// Mitsubishi GX Works2 project: אוטומציה 29.11 713   PLC: FX3G

// global labels: Global1
VAR_GLOBAL
  startDay AT X010 : BOOL;
  flourContainer AT D1110 : REAL;
  flourInput AT D1100 : REAL;
  yeastInput AT D1102 : REAL;
  yeatContainer AT D1112 : REAL;
  YeastContainer AT D1112 : REAL;
  waterInput AT D1104 : REAL;
  waterContainer AT D1114 : REAL;
  oilInput AT D1106 : REAL;
  oilContainer AT D1116 : REAL;
  spaicesInput AT D1108 : REAL;
  spaicesContainer AT D1118 : REAL;
  EmergencyStop AT X007 : BOOL;
  workDayLight AT Y010 : BOOL;
  endDay AT M8 : BOOL;
  outOfStock AT M7 : BOOL;
  startProduction AT M6 : BOOL;
END_VAR
VAR_GLOBAL CONSTANT
  minFlour : REAL := 100.0;
END_VAR
VAR_GLOBAL
  FlourOK AT M1 : BOOL;
END_VAR
VAR_GLOBAL CONSTANT
  fYratio : REAL := 0.2;
END_VAR
VAR_GLOBAL
  yeastOK AT M2 : BOOL;
END_VAR
VAR_GLOBAL CONSTANT
  wFratio : REAL := 0.5;
END_VAR
VAR_GLOBAL
  waterOK AT M3 : BOOL;
END_VAR
VAR_GLOBAL CONSTANT
  oFratio : REAL := 0.3;
END_VAR
VAR_GLOBAL
  oilOK AT M4 : BOOL;
END_VAR
VAR_GLOBAL CONSTANT
  sFratio : REAL := 0.1;
END_VAR
VAR_GLOBAL
  spaicesOK AT M5 : BOOL;
  LoadMaterialsButton AT X002 : BOOL;
  LoadMterialsLamp AT Y005 : BOOL;
END_VAR
VAR_GLOBAL CONSTANT
  flour_100 : REAL := 100;
  Yeast_20 : REAL := 20;
  water_50 : REAL := 50;
  oil_30 : REAL := 30;
  spices_10 : REAL := 10;
END_VAR
VAR_GLOBAL
  timeVal_3sec AT K30 : INT;
  prepTimer AT TC10 : BOOL;
  prepTimer_out AT TS10 : BOOL;
  startLisha AT X001 : BOOL;
  proofStartHatpaha AT M32 : BOOL;
  lishaMotor AT Y001 : BOOL;
  hatpaha_Counter AT CC1 : BOOL;
  doubleclick AT K2 : WORD;
  start_Hatpaha AT X011 : BOOL;
  outC1 AT CS1 : BOOL;
  y2timer AT TC22 : BOOL;
  TS22_out AT TS22 : BOOL;
  ind_blinkled AT M0 : BOOL;
  Hatpaha_led2 AT Y002 : BOOL;
  y3timer AT TC23 : BOOL;
  TS23_out AT TS23 : BOOL;
  Hatpaha_led3 AT Y003 : BOOL;
  hatpaha_timer AT TC32 : BOOL;
  TS32_OUT AT TS32 : BOOL;
  timeVal_BLINK AT K5 : INT;
  y4timer AT TC24 : BOOL;
  timeVal_4 AT K40 : INT;
  BAKE_LAMP AT Y004 : BOOL;
  TS24_out AT TS24 : BOOL;
  quality_check AT X003 : BOOL;
  Analog_Input_2 AT D8281 : INT;
  Save_analog_val AT D8201 : INT;
END_VAR
VAR_GLOBAL CONSTANT
  min_val : INT := 400;
  max_val : INT := 2000;
END_VAR
VAR_GLOBAL
  Analog_GT AT M11 : BOOL;
  Analog_LT AT M12 : BOOL;
  y6_timer AT TC26 : BOOL;
  timeVal_5 AT K50 : INT;
  TS26_out AT TS26 : BOOL;
  move_to_shelf_lamp AT Y006 : BOOL;
  check_counter AT CC2 : BOOL;
  double_check AT K2 : WORD;
  CC2_out AT CS2 : BOOL;
  batch_Rejact AT M23 : BOOL;
  in_Proportion AT M6 : BOOL;
END_VAR
VAR_GLOBAL CONSTANT
  iteration_Flour : INT := 100;
END_VAR
VAR_GLOBAL
  iteration_Flour_Container AT D1120 : REAL;
END_VAR
VAR_GLOBAL CONSTANT
  iteration_Flour_Amount : REAL := 100;
  iteration_Yeast_Amount : REAL := 20;
END_VAR
VAR_GLOBAL
  iteration_Yeast_Container AT D1122 : REAL;
END_VAR
VAR_GLOBAL CONSTANT
  iteration_Water_Amount : REAL := 50;
END_VAR
VAR_GLOBAL
  iteration_Water_Container AT D1124 : REAL;
END_VAR
VAR_GLOBAL CONSTANT
  iteration_Oil_Amount : REAL := 30;
END_VAR
VAR_GLOBAL
  iteration_Oil_Container AT D1126 : REAL;
END_VAR
VAR_GLOBAL CONSTANT
  iteration_Spices_Amount : REAL := 10;
END_VAR
VAR_GLOBAL
  iteration_Spices_Container AT D1128 : REAL;
  mearbel_container AT D1130 : REAL;
  hatpaha_Container AT D1132 : REAL;
  tavnit_bake_container AT D1134 : REAL;
  bakery_shelf_container AT D1136 : REAL;
  noFlour AT M40 : BOOL;
  noYeast AT M42 : BOOL;
  noWater AT M44 : BOOL;
  noOil AT M46 : BOOL;
  noSpices AT M48 : BOOL;
END_VAR
VAR_GLOBAL CONSTANT
  reset_0 : REAL;
END_VAR
VAR_GLOBAL
  finish_timer AT TC50 : BOOL;
  TS50_OUT AT TS50 : BOOL;
  ind_blinkled_finish AT M200 : BOOL;
  TS52_out AT TS52 : BOOL;
  TS54_out AT TS54 : BOOL;
  timeVal_BLINK2 AT K2 : INT;
  no_light_10 AT M60 : BOOL;
  end_day_light AT M62 : BOOL;
  ind AT M0 : BOOL;
  delete_mearbel AT M33 : BOOL;
  ind_move_to_tavnit AT M100 : BOOL;
  ind_move_to_bakery AT M102 : BOOL;
  y10blinkOn AT TC52 : BOOL;
  y10blinkOff AT TC54 : BOOL;
  y10_steady_light AT M70 : BOOL;
END_VAR
VAR_GLOBAL CONSTANT
  iteration_finished : REAL := 1;
END_VAR
VAR_GLOBAL
  ind_iteration_finished AT M250 : BOOL;
  ind_end_of_iteration AT M104 : BOOL;
  iteration_counter AT D1138 : REAL;
END_VAR
VAR_GLOBAL CONSTANT
  check_prev_lvl : REAL;
END_VAR
VAR_GLOBAL
  ind_first_lvl_finished AT M400 : BOOL;
  ind_X2_lvl_finished AT M402 : BOOL;
  ind_X11_lvl_finished AT M404 : BOOL;
END_VAR

// task Task_01 (event TRUE, interval 0, priority 31): POU_01

PROGRAM POU_01
(* structured ladder/FBD written out as ST: instructions are called as NAME(EN, inputs, outputs); _pN, _eN, _tN stand for wires *)
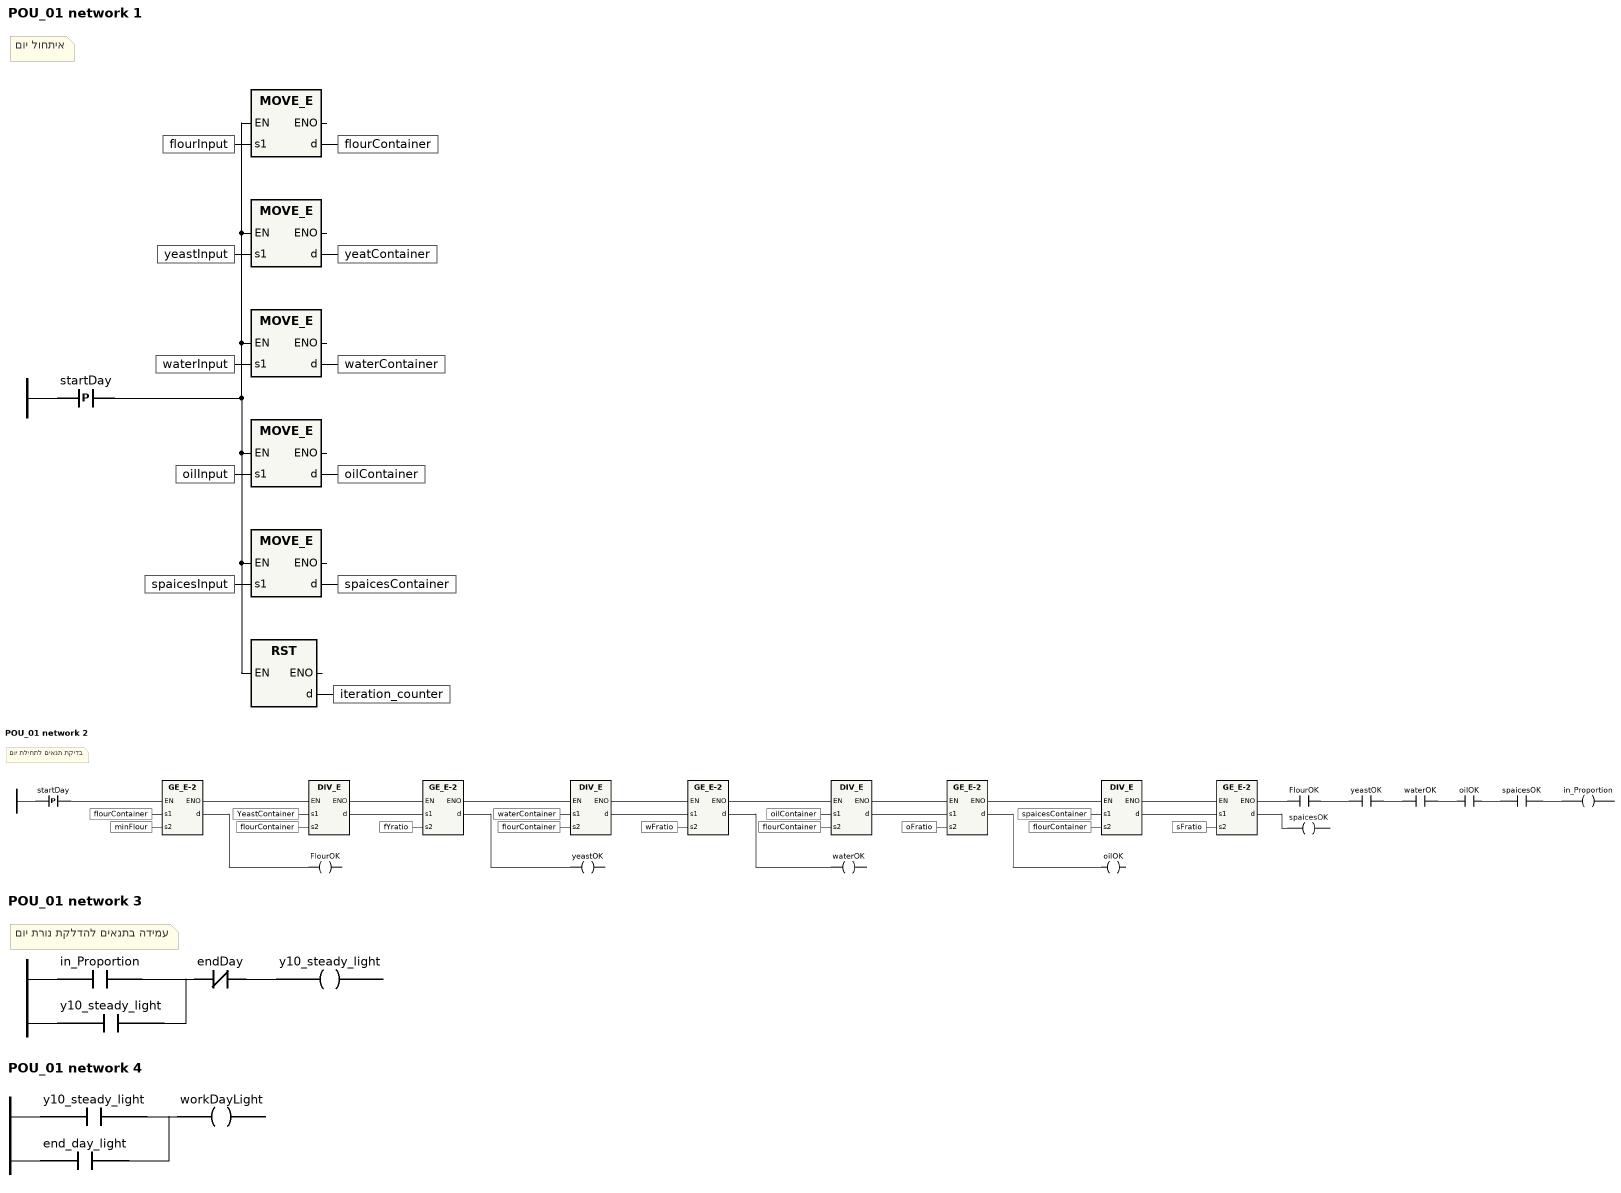
(* network 1 *)
(* איתחול יום *)
_p1 := LDP(TRUE, startDay);
MOVE_E(_p1, flourInput, flourContainer);
MOVE_E(_p1, yeastInput, yeatContainer);
MOVE_E(_p1, waterInput, waterContainer);
MOVE_E(_p1, oilInput, oilContainer);
MOVE_E(_p1, spaicesInput, spaicesContainer);
RST(_p1, iteration_counter);
(* network 2 *)
(* בדיקת תנאים לתחילת יום *)
_e2 := GE_E(LDP(TRUE, startDay), flourContainer, minFlour, _t1);
_e4 := DIV_E(_e2, YeastContainer, flourContainer, _t3);
_e6 := GE_E(_e4, _t3, fYratio, _t5);
_e8 := DIV_E(_e6, waterContainer, flourContainer, _t7);
_e10 := GE_E(_e8, _t7, wFratio, _t9);
_e12 := DIV_E(_e10, oilContainer, flourContainer, _t11);
_e14 := GE_E(_e12, _t11, oFratio, _t13);
_e16 := DIV_E(_e14, spaicesContainer, flourContainer, _t15);
_e18 := GE_E(_e16, _t15, sFratio, _t17);
in_Proportion := _e18 AND FlourOK AND yeastOK AND waterOK AND oilOK AND spaicesOK;
yeastOK := _t5;
waterOK := _t9;
oilOK := _t13;
spaicesOK := _t17;
FlourOK := _t1;
(* network 3 *)
(* עמידה בתנאים להדלקת נורת יום *)
y10_steady_light := (in_Proportion OR y10_steady_light) AND NOT endDay;
(* network 4 *)
workDayLight := y10_steady_light OR end_day_light;
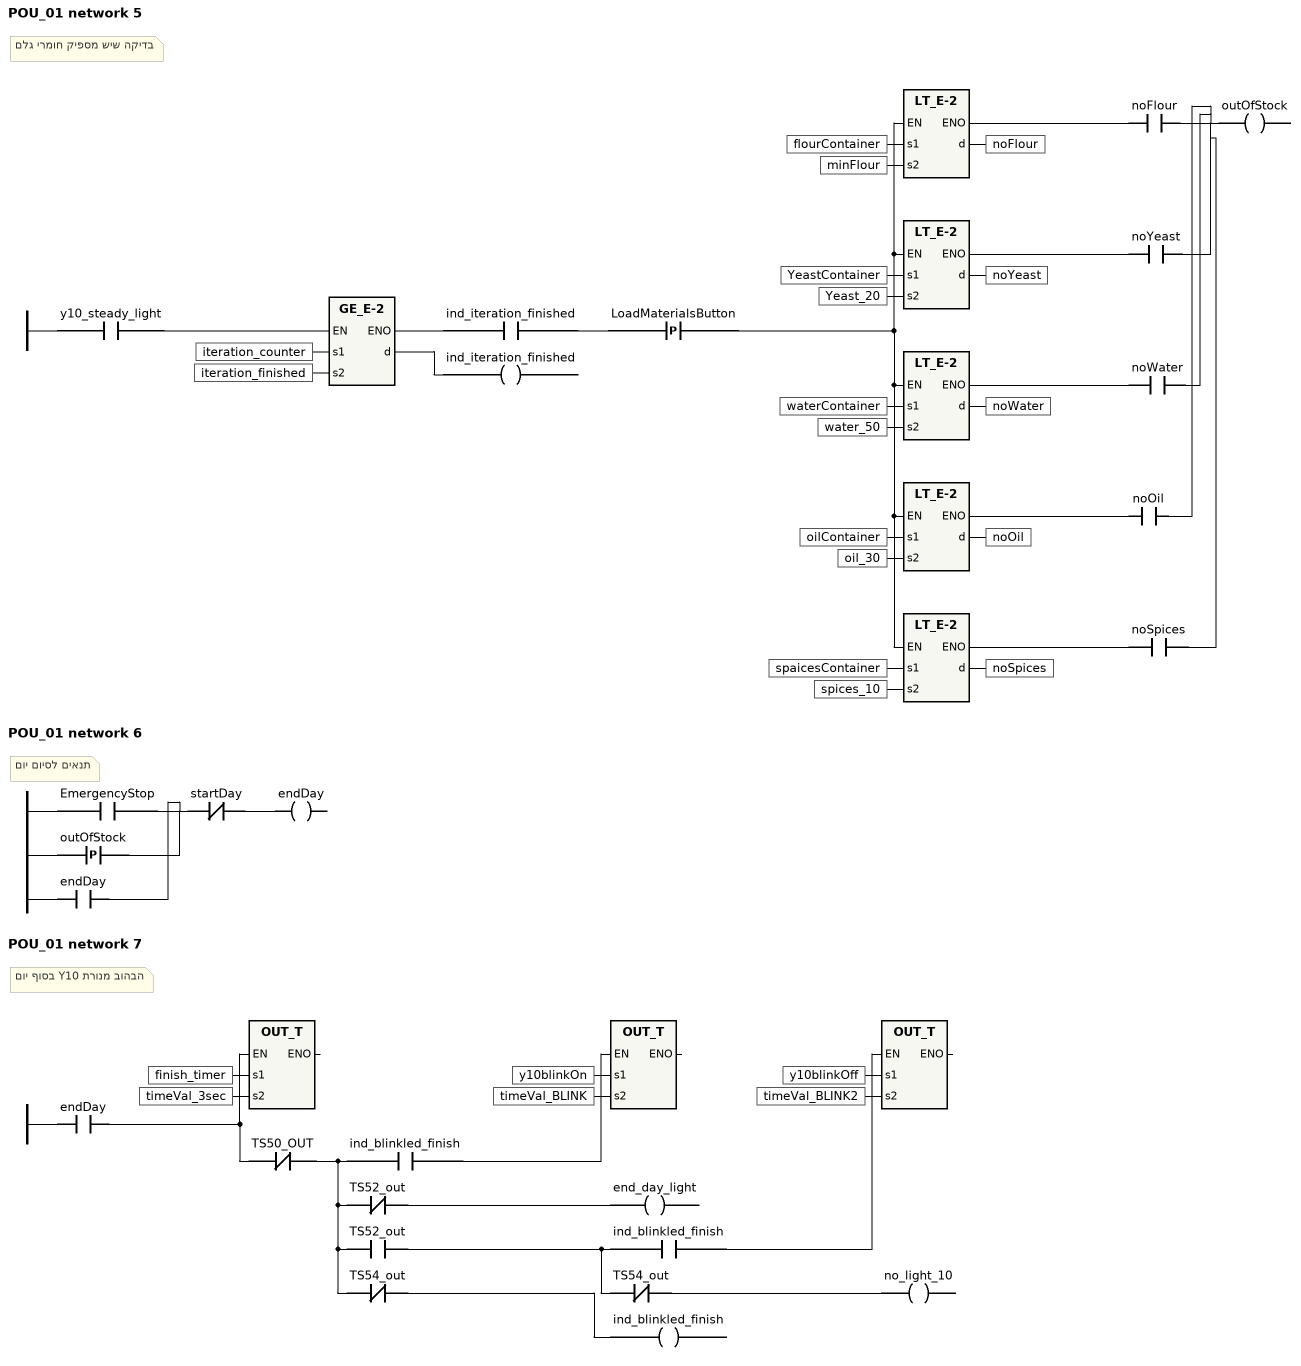
(* network 5 *)
(* בדיקה שיש מספיק חומרי גלם *)
_e2 := GE_E(y10_steady_light, iteration_counter, iteration_finished, _t1);
_p3 := _e2 AND ind_iteration_finished AND LDP(TRUE, LoadMaterialsButton);
_e4 := LT_E(_p3, flourContainer, minFlour, noFlour);
ind_iteration_finished := _t1;
_e5 := LT_E(_p3, YeastContainer, Yeast_20, noYeast);
_e6 := LT_E(_p3, waterContainer, water_50, noWater);
_e7 := LT_E(_p3, oilContainer, oil_30, noOil);
_e8 := LT_E(_p3, spaicesContainer, spices_10, noSpices);
outOfStock := (_e4 AND noFlour) OR (_e5 AND noYeast) OR (_e6 AND noWater) OR (_e7 AND noOil) OR (_e8 AND noSpices);
(* network 6 *)
(* תנאים לסיום יום *)
endDay := (EmergencyStop OR LDP(TRUE, outOfStock) OR endDay) AND NOT startDay;
(* network 7 *)
(* הבהוב מנורת Y10 בסוף יום *)
OUT_T(endDay, finish_timer, timeVal_3sec);
_p1 := endDay AND NOT TS50_OUT;
OUT_T(_p1 AND ind_blinkled_finish, y10blinkOn, timeVal_BLINK);
end_day_light := _p1 AND NOT TS52_out;
_p2 := _p1 AND TS52_out;
OUT_T(_p2 AND ind_blinkled_finish, y10blinkOff, timeVal_BLINK2);
no_light_10 := _p2 AND NOT TS54_out;
ind_blinkled_finish := _p1 AND NOT TS54_out;
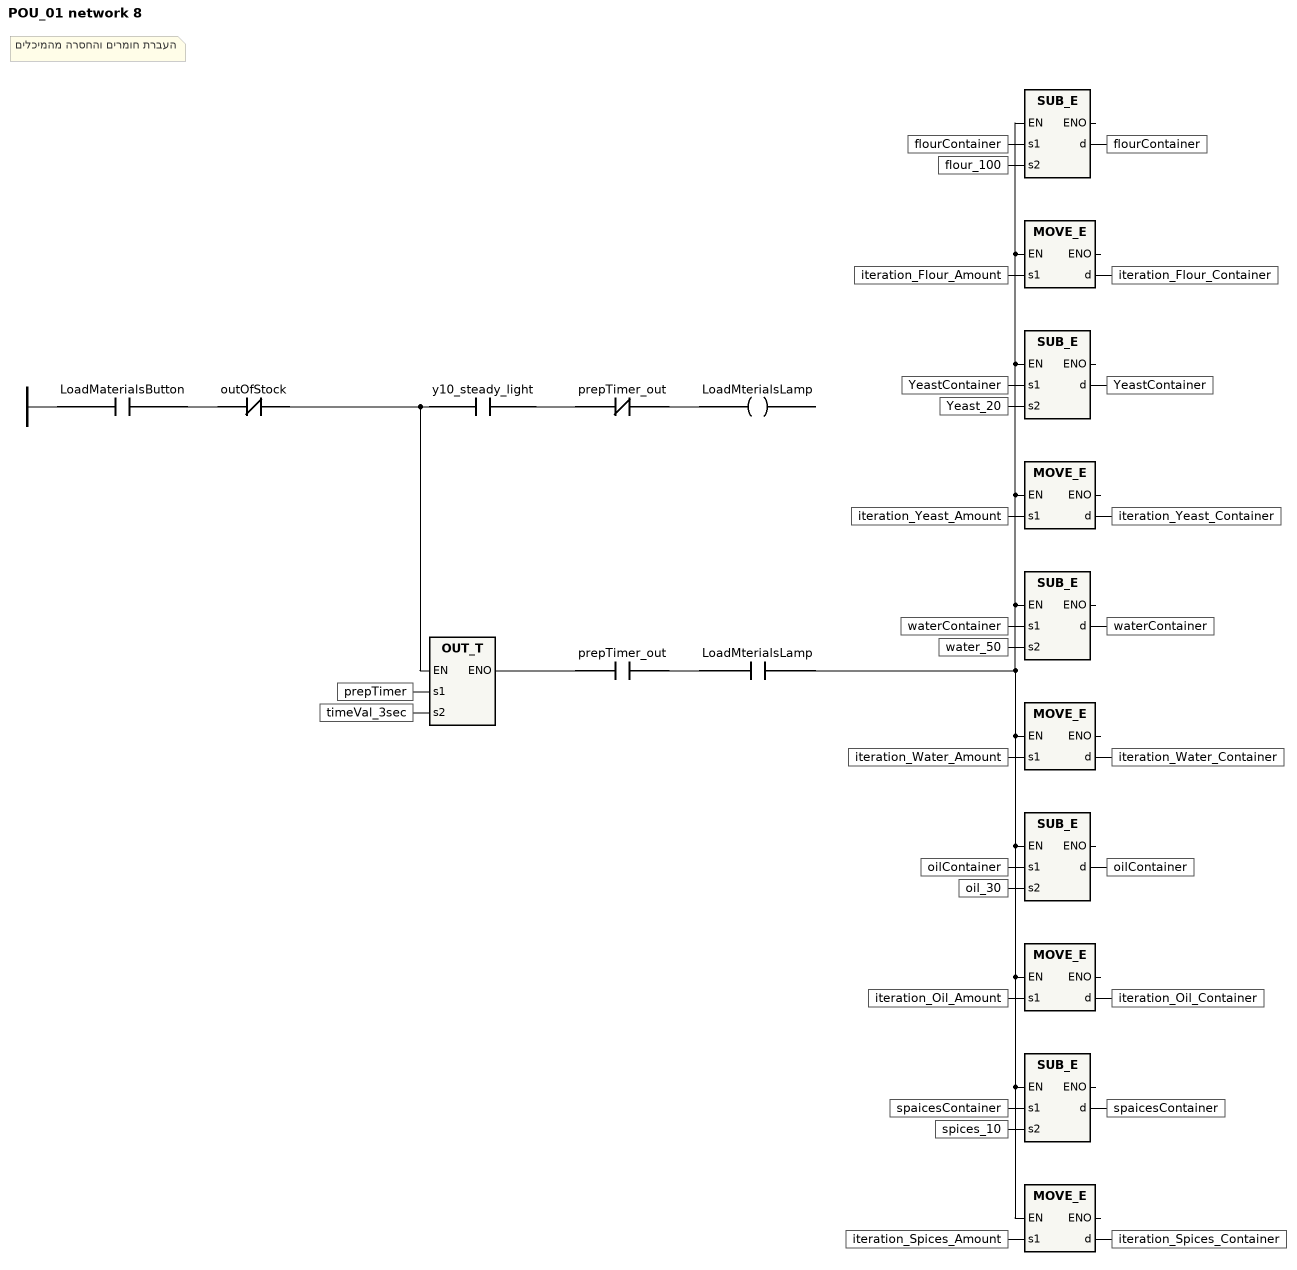
(* network 8 *)
(* העברת חומרים והחסרה מהמיכלים *)
_p1 := LoadMaterialsButton AND NOT outOfStock;
_e2 := OUT_T(_p1, prepTimer, timeVal_3sec);
_p3 := _e2 AND prepTimer_out AND LoadMterialsLamp;
SUB_E(_p3, flourContainer, flour_100, flourContainer);
MOVE_E(_p3, iteration_Flour_Amount, iteration_Flour_Container);
SUB_E(_p3, YeastContainer, Yeast_20, YeastContainer);
LoadMterialsLamp := _p1 AND y10_steady_light AND NOT prepTimer_out;
MOVE_E(_p3, iteration_Yeast_Amount, iteration_Yeast_Container);
SUB_E(_p3, waterContainer, water_50, waterContainer);
MOVE_E(_p3, iteration_Water_Amount, iteration_Water_Container);
SUB_E(_p3, oilContainer, oil_30, oilContainer);
MOVE_E(_p3, iteration_Oil_Amount, iteration_Oil_Container);
SUB_E(_p3, spaicesContainer, spices_10, spaicesContainer);
MOVE_E(_p3, iteration_Spices_Amount, iteration_Spices_Container);
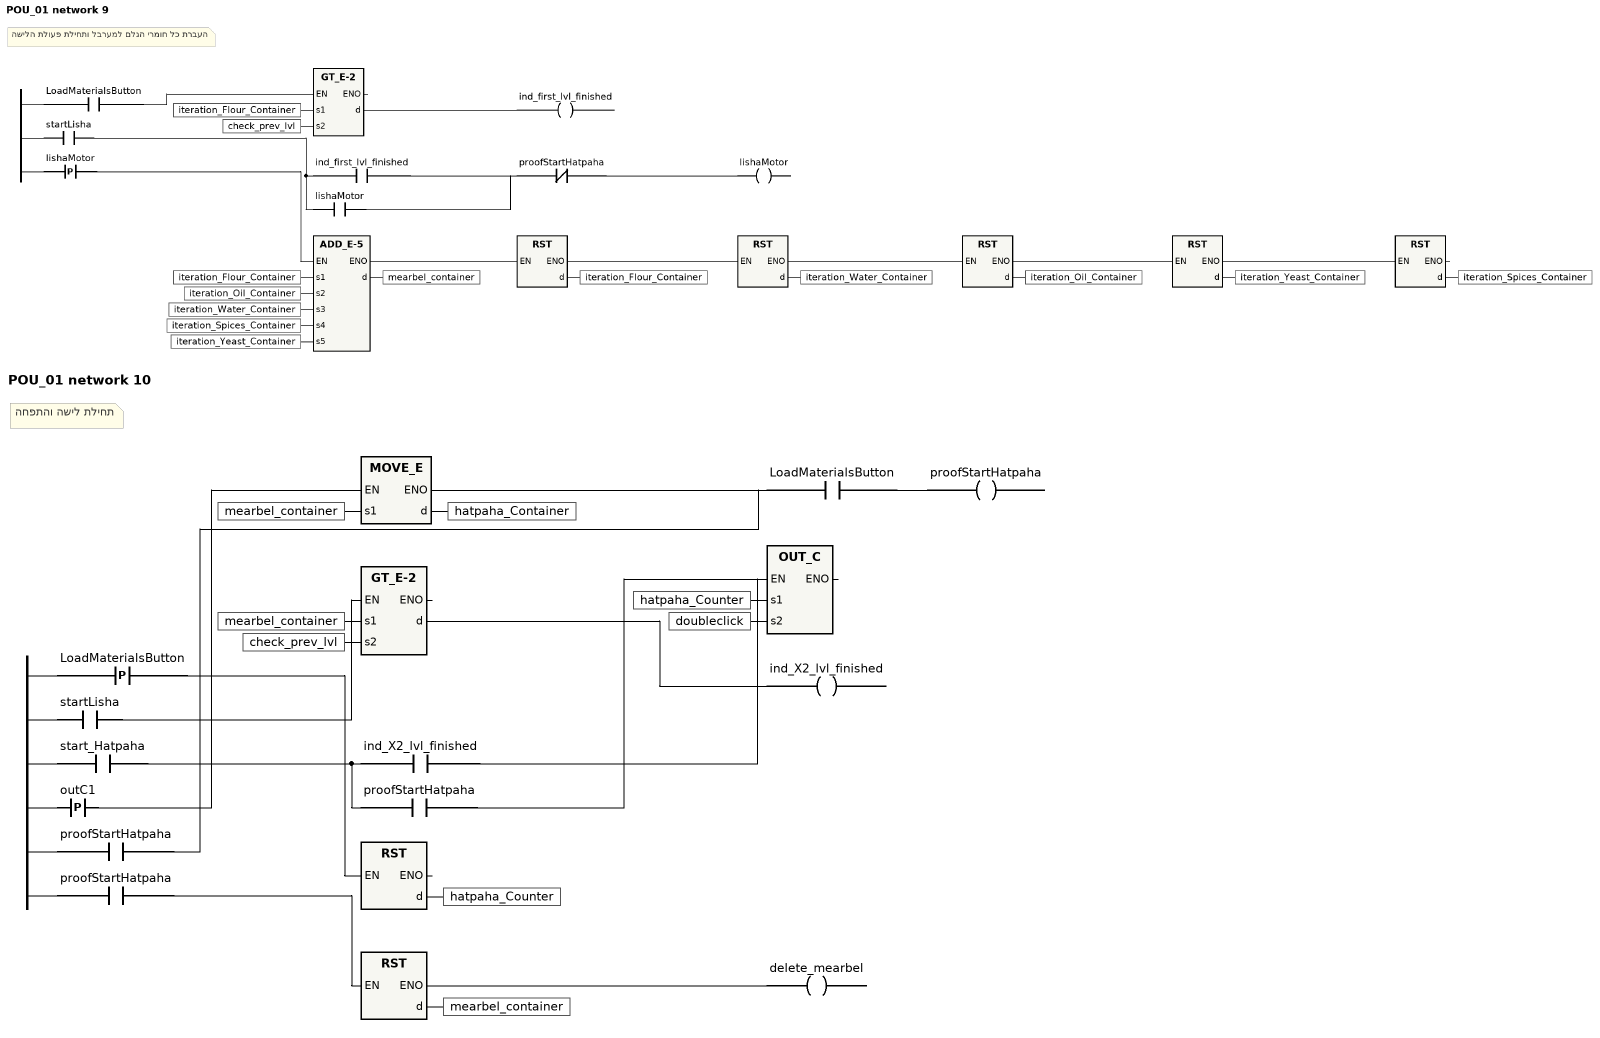
(* network 9 *)
(* העברת כל חומרי הגלם למערבל ותחילת פעולת הלישה *)
GT_E(LoadMaterialsButton, iteration_Flour_Container, check_prev_lvl, _t1);
ind_first_lvl_finished := _t1;
lishaMotor := ((startLisha AND ind_first_lvl_finished) OR (startLisha AND lishaMotor)) AND NOT proofStartHatpaha;
_e2 := ADD_E(LDP(TRUE, lishaMotor), iteration_Flour_Container, iteration_Oil_Container, iteration_Water_Container, iteration_Spices_Container, iteration_Yeast_Container, mearbel_container);
_e3 := RST(_e2, iteration_Flour_Container);
_e4 := RST(_e3, iteration_Water_Container);
_e5 := RST(_e4, iteration_Oil_Container);
_e6 := RST(_e5, iteration_Yeast_Container);
RST(_e6, iteration_Spices_Container);
(* network 10 *)
(* תחילת לישה והתפחה *)
RST(LDP(TRUE, LoadMaterialsButton), hatpaha_Counter);
GT_E(startLisha, mearbel_container, check_prev_lvl, _t1);
ind_X2_lvl_finished := _t1;
OUT_C((start_Hatpaha AND ind_X2_lvl_finished) OR (start_Hatpaha AND proofStartHatpaha), hatpaha_Counter, doubleclick);
_e2 := MOVE_E(LDP(TRUE, outC1), mearbel_container, hatpaha_Container);
proofStartHatpaha := (_e2 OR proofStartHatpaha) AND LoadMaterialsButton;
_e3 := RST(proofStartHatpaha, mearbel_container);
delete_mearbel := _e3;
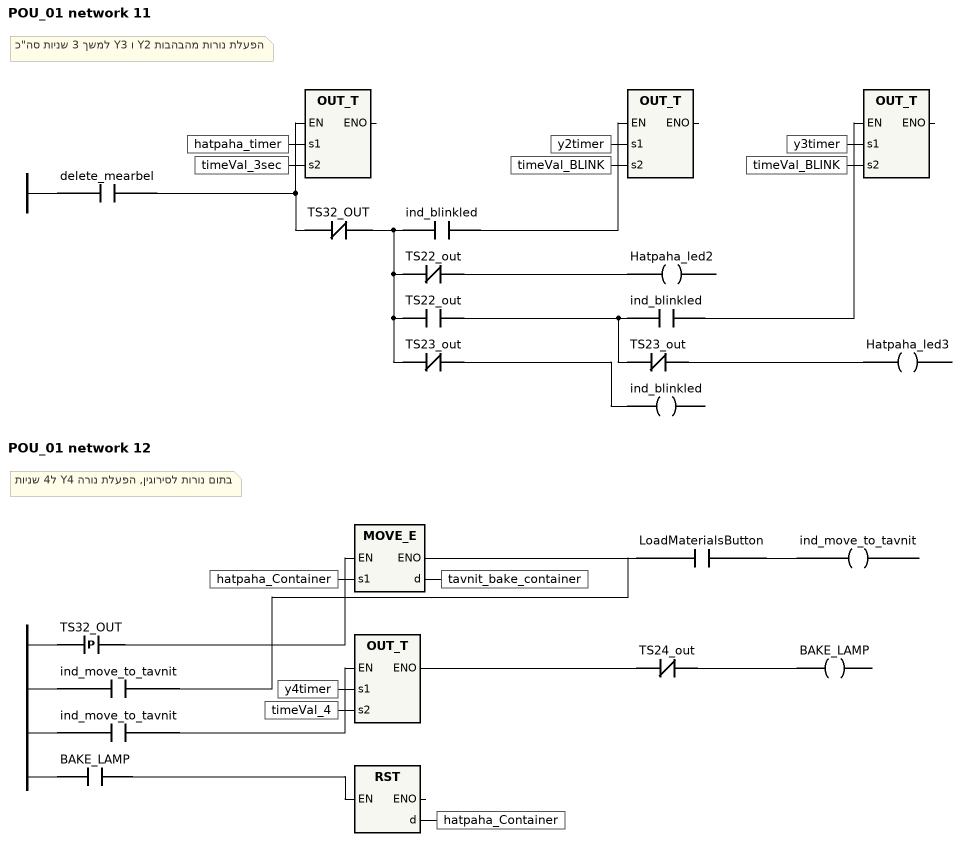
(* network 11 *)
(* הפעלת נורות מהבהבות Y2 ו Y3 למשך 3 שניות סה"כ *)
OUT_T(delete_mearbel, hatpaha_timer, timeVal_3sec);
_p1 := delete_mearbel AND NOT TS32_OUT;
OUT_T(_p1 AND ind_blinkled, y2timer, timeVal_BLINK);
Hatpaha_led2 := _p1 AND NOT TS22_out;
_p2 := _p1 AND TS22_out;
OUT_T(_p2 AND ind_blinkled, y3timer, timeVal_BLINK);
Hatpaha_led3 := _p2 AND NOT TS23_out;
ind_blinkled := _p1 AND NOT TS23_out;
(* network 12 *)
(* בתום נורות לסירוגין, הפעלת נורה Y4 ל4 שניות *)
_e1 := MOVE_E(LDP(TRUE, TS32_OUT), hatpaha_Container, tavnit_bake_container);
ind_move_to_tavnit := (_e1 OR ind_move_to_tavnit) AND LoadMaterialsButton;
_e2 := OUT_T(ind_move_to_tavnit, y4timer, timeVal_4);
BAKE_LAMP := _e2 AND NOT TS24_out;
RST(BAKE_LAMP, hatpaha_Container);
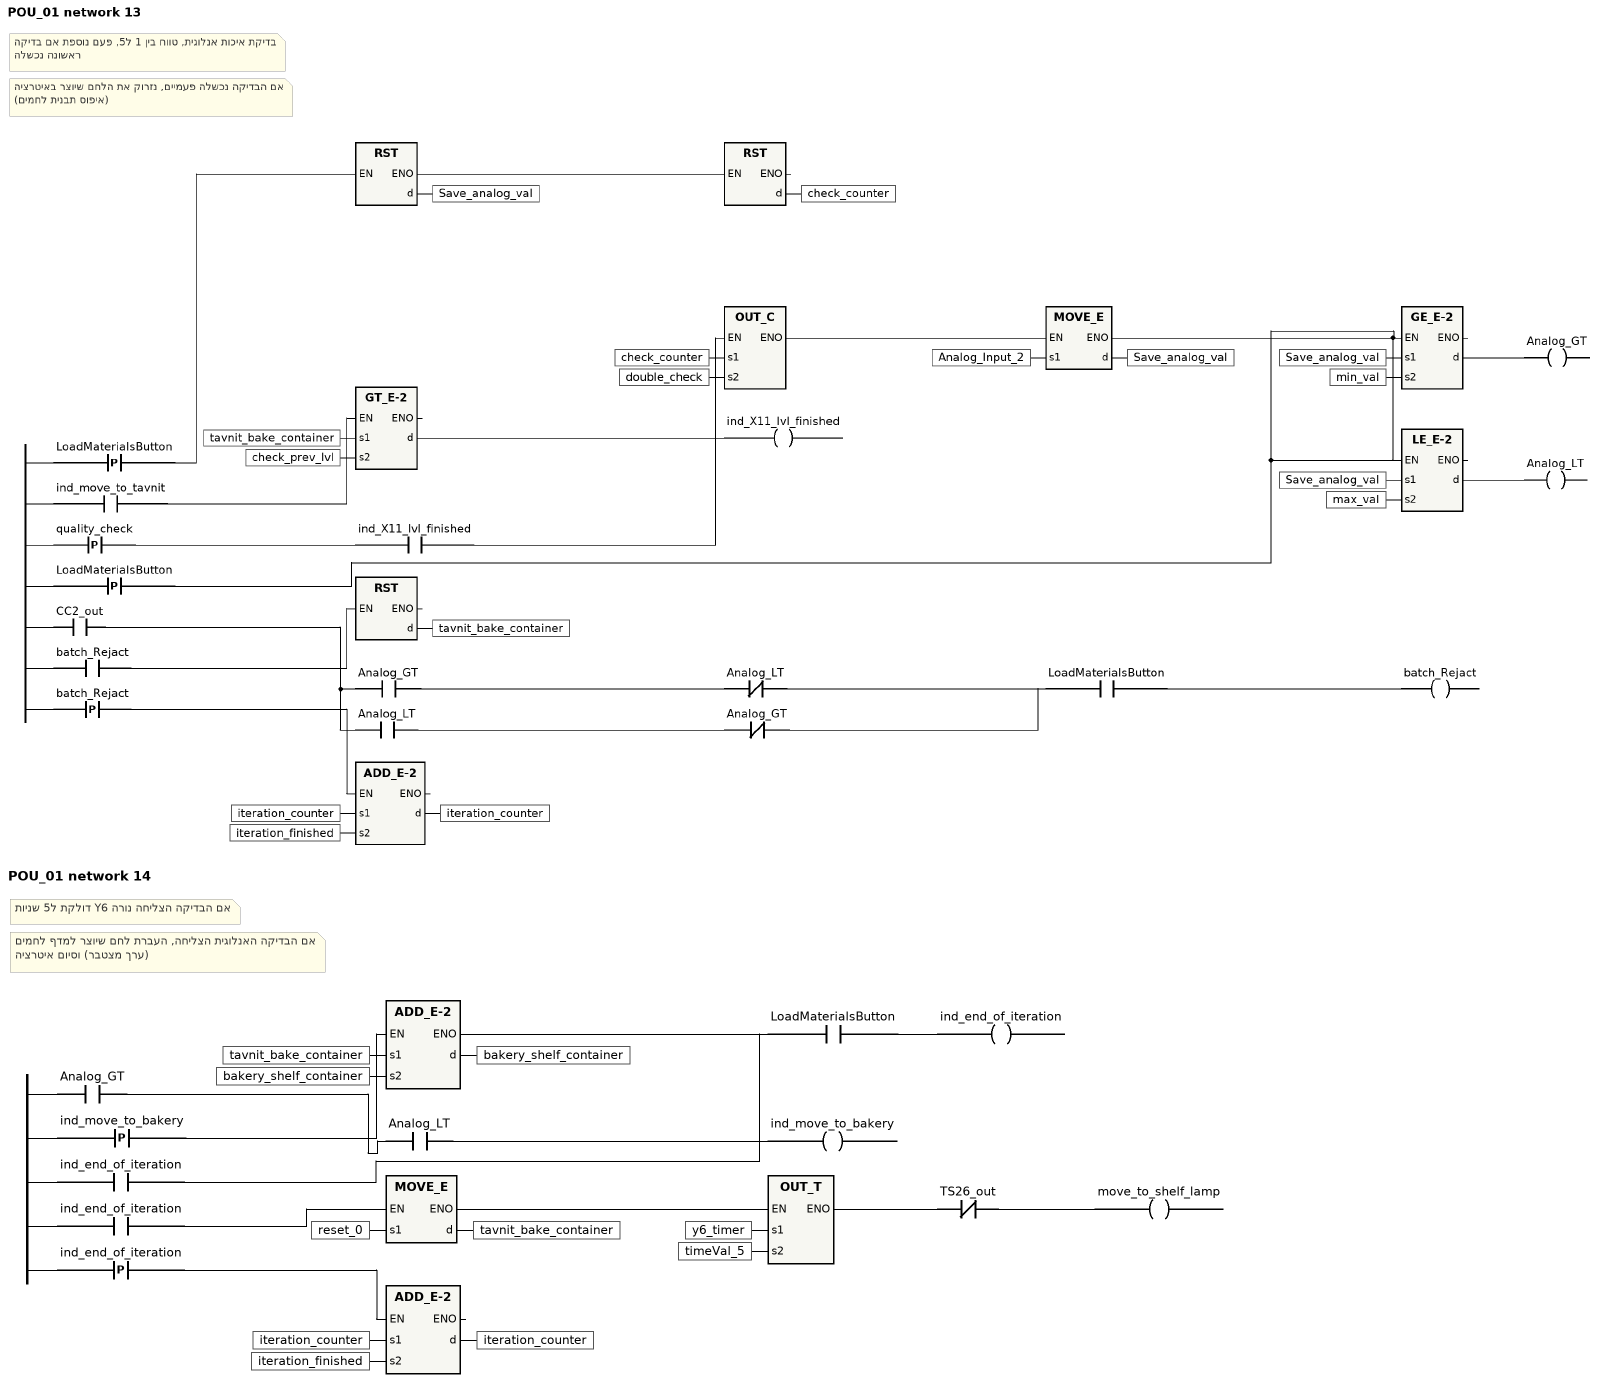
(* network 13 *)
(* בדיקת איכות אנלוגית, טווח בין 1 ל5, פעם נוספת אם בדיקה ראשונה נכשלה *)
(* אם הבדיקה נכשלה פעמיים, נזרוק את הלחם שיוצר באיטרציה (איפוס תבנית לחמים) *)
_e1 := RST(LDP(TRUE, LoadMaterialsButton), Save_analog_val);
RST(_e1, check_counter);
GT_E(ind_move_to_tavnit, tavnit_bake_container, check_prev_lvl, _t2);
ind_X11_lvl_finished := _t2;
_e3 := OUT_C(LDP(TRUE, quality_check) AND ind_X11_lvl_finished, check_counter, double_check);
_e4 := MOVE_E(_e3, Analog_Input_2, Save_analog_val);
_p5 := _e4 OR LDP(TRUE, LoadMaterialsButton);
GE_E(_p5, Save_analog_val, min_val, _t6);
Analog_GT := _t6;
LE_E(_p5, Save_analog_val, max_val, _t7);
Analog_LT := _t7;
batch_Rejact := ((CC2_out AND Analog_GT AND NOT Analog_LT) OR (CC2_out AND Analog_LT AND NOT Analog_GT)) AND LoadMaterialsButton;
RST(batch_Rejact, tavnit_bake_container);
ADD_E(LDP(TRUE, batch_Rejact), iteration_counter, iteration_finished, iteration_counter);
(* network 14 *)
(* אם הבדיקה הצליחה נורה Y6 דולקת ל5 שניות *)
(* אם הבדיקה האנלוגית הצליחה, העברת לחם שיוצר למדף לחמים (ערך מצטבר) וסיום איטרציה *)
ind_move_to_bakery := Analog_GT AND Analog_LT;
_e1 := ADD_E(LDP(TRUE, ind_move_to_bakery), tavnit_bake_container, bakery_shelf_container, bakery_shelf_container);
ind_end_of_iteration := (_e1 OR ind_end_of_iteration) AND LoadMaterialsButton;
_e2 := MOVE_E(ind_end_of_iteration, reset_0, tavnit_bake_container);
_e3 := OUT_T(_e2, y6_timer, timeVal_5);
move_to_shelf_lamp := _e3 AND NOT TS26_out;
ADD_E(LDP(TRUE, ind_end_of_iteration), iteration_counter, iteration_finished, iteration_counter);
END_PROGRAM
